# EPICS autosave request: ADApp/Db/NDGather_settings.req
file "NDPluginBase_settings.req", P=$(P), R=$(R)
$(P)$(R)SortTime
$(P)$(R)SortMode
